TYPE M2ConstantsTiltX :
STRUCT
	///Motor reduction ratio
	MOT_TO_RED_RATIO: LREAL := 1526.0;
	///Transmission ratio between the motor reduction and the screw
	RED_TO_SCREW_RATIO: LREAL := 2.0;
	///Transmission ratio between the potentiometer and the screw
	SCREW_TO_POT_RATIO: LREAL := 0.5;
	///Minimum position of the axis, in micrometer
	MIN_POSITION: LREAL := 260.0;
	///Maximum position of the axis, in micrometer
	MAX_POSITION: LREAL := 1200.0;
	///Screw pitch, in micrometer
	SCREW_PITCH: LREAL := 1000.0;
	///Motor feedback resolution (pulses per revolution of the motor rotor)
	FEEDBACK_RESOLUTION: LREAL := 3;
	///Max number of revolutions of the potentiometer
	POTENTIOMETER_REVOLUTIONS: LREAL := 3;
END_STRUCT
END_TYPE

(* stored: Version 1.1.0.1, ProductVersion 3.1.4019.2
   DUT M2ConstantsTiltX: Id {8a8ba1ed-b610-4c39-ac1d-71bbf942b09d} *)
